FUNCTION EqualsRange : BOOL
VAR_INPUT
	range1 : Range;
	range2 : Range;
	epsilon : LREAL;
END_VAR

EqualsRange := EqualsLREAL(range1.Bottom, range2.Bottom, epsilon)
			AND EqualsLREAL(range1.Top, range2.Top, epsilon);

END_FUNCTION

(* stored: Version 1.1.0.1
   POU EqualsRange: Id {bf5b60eb-5b53-0f64-3dc8-e3bca8b3d687}, SpecialFunc None *)
